// return the bIn as passed. set the value to FALSE.
FUNCTION F_Gate : BOOL
VAR_IN_OUT
	bIn : BOOL;
END_VAR

F_Gate := bIn;
// reset if true. (below is equivalent of IF bIn THEN bIn := FALSE; END_IF)
bIn := FALSE;

END_FUNCTION

(* stored: Version 1.1.0.1, ProductVersion 3.1.4020.12
   POU F_Gate: Id {97b3a654-cb47-4f65-b0a1-b8a5603611a0}, SpecialFunc None *)
